// TIA Portal project "Water_Tank_For_Exam" (V12)

(* hardware
DEVICE "S7-1200 station_1"  SIMATIC 1200-Station
   slot 0: "S7-1200 rack"  Rack  V1.0
   slot 1: "Water_Tank_Logic"  CPU 1211C DC/DC/DC  6ES7 211-1AE31-0XB0  V3.0
DEVICE "S7-1500 station_1"  S7-1500 station
   slot 0: "Rail_0"  6ES7 590-1***0-0AA0
   slot 1: "PLC_1"  CPU 1513-1 PN  6ES7 513-1AL00-0AB0  V1.0
   slot 2: "DI 16x24VDC HF_1"  DI 16x24VDC HF  6ES7 521-1BH00-0AB0  V1.0
   slot 3: "DQ 8x24VDC/2A HF_1"  DQ 8x24VDC/2A HF  6ES7 522-1BF00-0AB0  V1.0
*)

// ===== PLC "Water_Tank_Logic"  CPU 1211C DC/DC/DC =====

VAR_GLOBAL   // PLC tag table "Default tag table"
   "GreenValveOpenLED" AT %Q0.0 : Bool;
   "redTankEmpty" AT %Q0.1 : Bool;
   "YellowTankFull" AT %Q0.2 : Bool;
   "LowSensor" AT %I0.0 : Bool;
   "HighLSensor" AT %I0.1 : Bool;
   "Manual" AT %I0.2 : Bool;
   "start" AT %I0.3 : Bool;
   "detectContainer" AT %I0.4 : Bool;
   "waterValve" AT %Q0.4 : Bool;
   "lacth" AT %M0.0 : Bool;
   "OpenValvePB" AT %I0.5 : Bool;
   "flashingEmptyLED" AT %Q0.3 : Bool;
   "autoMode" AT %I0.6 : Bool;
   "Counter5Mem" AT %M100.1 : Bool;
   "TimerFlash" AT %M100.0 : Bool;
   "Tag_1" AT %M100.2 : Bool;
END_VAR

// folder: System blocks/Program resources

DATA_BLOCK "IEC_Timer_0_DB"   // DB1
{ S7_Optimized_Access := 'FALSE' }
AUTHOR : Simatic
FAMILY : IEC
NAME : IEC_TMR
VERSION : 1.0
// stored: InstanceOfName ?
"?"
BEGIN
END_DATA_BLOCK

DATA_BLOCK "Counter_5"   // DB2
{ S7_Optimized_Access := 'FALSE' }
AUTHOR : Simatic
FAMILY : IEC
NAME : CNTR
VERSION : 1.0
// stored: InstanceOfName ?
"?"
BEGIN
END_DATA_BLOCK

DATA_BLOCK "Water_Running_timer"   // DB3
{ S7_Optimized_Access := 'FALSE' }
AUTHOR : Simatic
FAMILY : IEC
NAME : IEC_TMR
VERSION : 1.0
// stored: InstanceOfName ?
"?"
BEGIN
END_DATA_BLOCK

DATA_BLOCK "water_Still_in_Tank"   // DB4
{ S7_Optimized_Access := 'FALSE' }
AUTHOR : Simatic
FAMILY : IEC
NAME : IEC_TMR
VERSION : 1.0
// stored: InstanceOfName ?
"?"
BEGIN
END_DATA_BLOCK

DATA_BLOCK "Valve_counter"   // DB5
{ S7_Optimized_Access := 'FALSE' }
AUTHOR : Simatic
FAMILY : IEC
NAME : CNTR
VERSION : 1.0
// stored: InstanceOfName ?
"?"
BEGIN
END_DATA_BLOCK

DATA_BLOCK "Pulsating"   // DB7
{ S7_Optimized_Access := 'FALSE' }
AUTHOR : Simatic
FAMILY : IEC
NAME : IEC_TMR
VERSION : 1.0
// stored: InstanceOfName ?
"?"
BEGIN
END_DATA_BLOCK

DATA_BLOCK "Water_Valve_Timer"   // DB8
{ S7_Optimized_Access := 'FALSE' }
AUTHOR : Simatic
FAMILY : IEC
NAME : IEC_TMR
VERSION : 1.0
// stored: InstanceOfName ?
"?"
BEGIN
END_DATA_BLOCK

DATA_BLOCK "Water_remaining_timer"   // DB9
{ S7_Optimized_Access := 'FALSE' }
AUTHOR : Simatic
FAMILY : IEC
NAME : IEC_TMR
VERSION : 1.0
// stored: InstanceOfName ?
"?"
BEGIN
END_DATA_BLOCK

// folder: (top level)

FUNCTION "Water_Tank_Status_And_Control" : Void   // FC1, LAD
{ S7_Optimized_Access := 'FALSE' }
VERSION : 0.1
BEGIN

REGION Network 1: LED to indicate a low tank
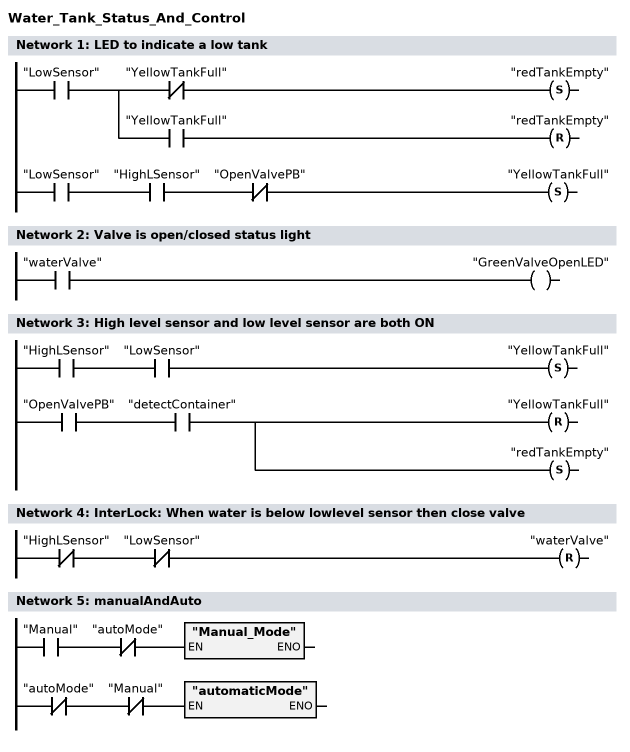
   RUNG wire#powerrail
      Contact( "LowSensor" )
      wire#w1
      I_Contact( "YellowTankFull" )
      S_Coil( "redTankEmpty" )
   END_RUNG
   RUNG wire#w1
      Contact( "YellowTankFull" )
      R_Coil( "redTankEmpty" )
   END_RUNG
   RUNG wire#powerrail
      Contact( "LowSensor" )
      Contact( "HighLSensor" )
      I_Contact( "OpenValvePB" )
      S_Coil( "YellowTankFull" )
   END_RUNG
   // the same network as SCL:
   IF "LowSensor" AND NOT "YellowTankFull" THEN "redTankEmpty" := TRUE; END_IF;
   IF "LowSensor" AND "YellowTankFull" THEN "redTankEmpty" := FALSE; END_IF;
   IF "LowSensor" AND "HighLSensor" AND NOT "OpenValvePB" THEN "YellowTankFull" := TRUE; END_IF;
END_REGION

REGION Network 2: Valve is open/closed status light
   RUNG wire#powerrail
      Contact( "waterValve" )
      Coil( "GreenValveOpenLED" )
   END_RUNG
   // the same network as SCL:
   "GreenValveOpenLED" := "waterValve";
END_REGION

REGION Network 3: High level sensor and low level sensor are both ON
   RUNG wire#powerrail
      Contact( "HighLSensor" )
      Contact( "LowSensor" )
      S_Coil( "YellowTankFull" )
   END_RUNG
   RUNG wire#powerrail
      Contact( "OpenValvePB" )
      Contact( "detectContainer" )
      wire#w1
      R_Coil( "YellowTankFull" )
   END_RUNG
   RUNG wire#w1
      S_Coil( "redTankEmpty" )
   END_RUNG
   // the same network as SCL:
   IF "HighLSensor" AND "LowSensor" THEN "YellowTankFull" := TRUE; END_IF;
   IF "OpenValvePB" AND "detectContainer" THEN
       "YellowTankFull" := FALSE;
       "redTankEmpty" := TRUE;
   END_IF;
END_REGION

REGION Network 4: InterLock: When water is below lowlevel sensor then close valve
   RUNG wire#powerrail
      I_Contact( "HighLSensor" )
      I_Contact( "LowSensor" )
      R_Coil( "waterValve" )
   END_RUNG
   // the same network as SCL:
   IF NOT "HighLSensor" AND NOT "LowSensor" THEN "waterValve" := FALSE; END_IF;
END_REGION

REGION Network 5: manualAndAuto
   RUNG wire#powerrail
      Contact( "Manual" )
      I_Contact( "autoMode" )
      "Manual_Mode"()
   END_RUNG
   RUNG wire#powerrail
      I_Contact( "autoMode" )
      I_Contact( "Manual" )
      "automaticMode"()
   END_RUNG
   // the same network as SCL:
   IF "Manual" AND NOT "autoMode" THEN "Manual_Mode"(); END_IF;
   IF NOT "autoMode" AND NOT "Manual" THEN "automaticMode"(); END_IF;
END_REGION
END_FUNCTION

FUNCTION "Manual_Mode" : Void   // FC2, LAD
{ S7_Optimized_Access := 'FALSE' }
VERSION : 0.1
   VAR_TEMP   // added for the SCL form of the ladder/FBD networks
      _w1 : Bool;
   END_VAR
BEGIN

REGION Network 1: manual mode
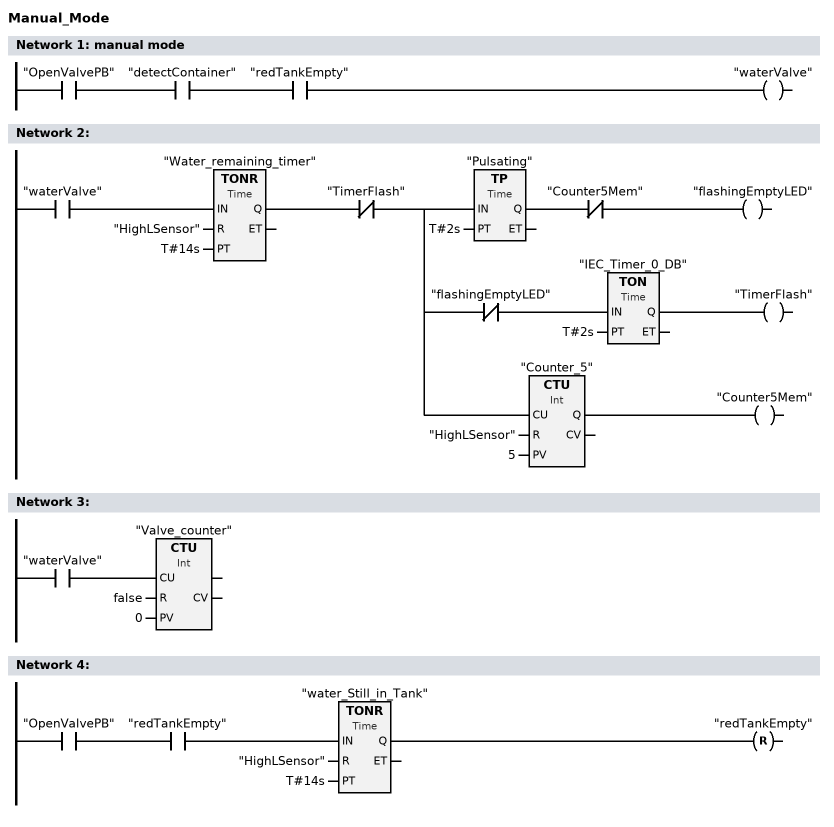
   RUNG wire#powerrail
      Contact( "OpenValvePB" )
      Contact( "detectContainer" )
      Contact( "redTankEmpty" )
      Coil( "waterValve" )
   END_RUNG
   // the same network as SCL:
   "waterValve" := "OpenValvePB" AND "detectContainer" AND "redTankEmpty";
END_REGION

REGION Network 2
   "Water_remaining_timer".TONR(IN := "waterValve", R := "HighLSensor", PT := T#14s);
   #_w1 := "Water_remaining_timer".Q AND NOT "TimerFlash";
   "Pulsating".TP(IN := #_w1, PT := T#2s);
   "flashingEmptyLED" := "Pulsating".Q AND NOT "Counter5Mem";
   "IEC_Timer_0_DB".TON(IN := #_w1 AND NOT "flashingEmptyLED", PT := T#2s);
   "TimerFlash" := "IEC_Timer_0_DB".Q;
   "Counter_5".CTU(CU := #_w1, R := "HighLSensor", PV := 5);
   "Counter5Mem" := "Counter_5".Q;
END_REGION

REGION Network 3
   "Valve_counter".CTU(CU := "waterValve", R := false, PV := 0);
END_REGION

REGION Network 4
   "water_Still_in_Tank".TONR(IN := "OpenValvePB" AND "redTankEmpty", R := "HighLSensor", PT := T#14s);
   IF "water_Still_in_Tank".Q THEN "redTankEmpty" := FALSE; END_IF;
END_REGION
END_FUNCTION

FUNCTION "automaticMode" : Void   // FC3, LAD
{ S7_Optimized_Access := 'FALSE' }
VERSION : 0.1
   VAR_TEMP   // added for the SCL form of the ladder/FBD networks
      _w1 : Bool;
   END_VAR
BEGIN

REGION Network 1: Automode Detects the container
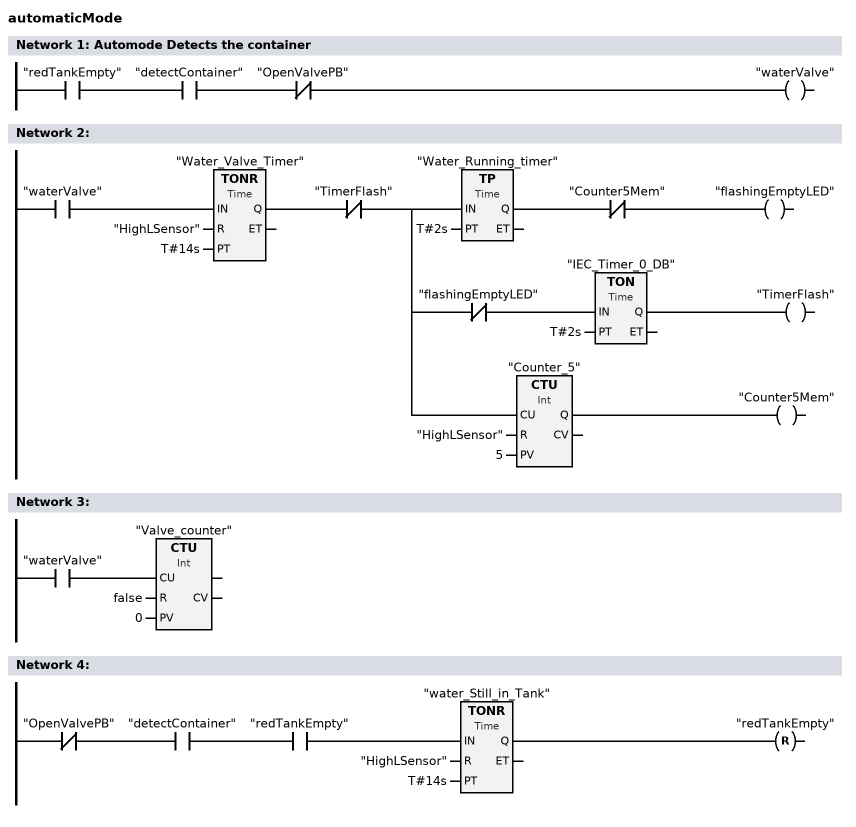
   RUNG wire#powerrail
      Contact( "redTankEmpty" )
      Contact( "detectContainer" )
      I_Contact( "OpenValvePB" )
      Coil( "waterValve" )
   END_RUNG
   // the same network as SCL:
   "waterValve" := "redTankEmpty" AND "detectContainer" AND NOT "OpenValvePB";
END_REGION

REGION Network 2
   "Water_Valve_Timer".TONR(IN := "waterValve", R := "HighLSensor", PT := T#14s);
   #_w1 := "Water_Valve_Timer".Q AND NOT "TimerFlash";
   "Water_Running_timer".TP(IN := #_w1, PT := T#2s);
   "flashingEmptyLED" := "Water_Running_timer".Q AND NOT "Counter5Mem";
   "IEC_Timer_0_DB".TON(IN := #_w1 AND NOT "flashingEmptyLED", PT := T#2s);
   "TimerFlash" := "IEC_Timer_0_DB".Q;
   "Counter_5".CTU(CU := #_w1, R := "HighLSensor", PV := 5);
   "Counter5Mem" := "Counter_5".Q;
END_REGION

REGION Network 3
   "Valve_counter".CTU(CU := "waterValve", R := false, PV := 0);
END_REGION

REGION Network 4
   "water_Still_in_Tank".TONR(IN := NOT "OpenValvePB" AND "detectContainer" AND "redTankEmpty",
                           R := "HighLSensor",
                           PT := T#14s);
   IF "water_Still_in_Tank".Q THEN "redTankEmpty" := FALSE; END_IF;
END_REGION
END_FUNCTION

ORGANIZATION_BLOCK "Main"   // OB1, LAD, ProgramCycle
TITLE = "Main Program Sweep (Cycle)"
{ S7_Optimized_Access := 'FALSE' }
VERSION : 0.1
   VAR_TEMP   // added for the SCL form of the ladder/FBD networks
      _w1 : Bool;
   END_VAR
BEGIN

REGION Network 1: Start and Stop the Whole plant
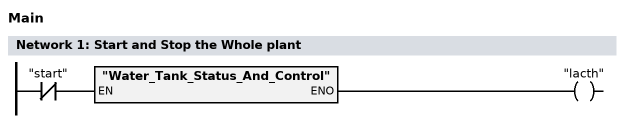
   RUNG wire#powerrail
      I_Contact( "start" )
      "Water_Tank_Status_And_Control"()
      Coil( "lacth" )
   END_RUNG
   // the same network as SCL:
   "Water_Tank_Status_And_Control"(EN := NOT "start", ENO => #_w1);
   "lacth" := #_w1;
END_REGION
END_ORGANIZATION_BLOCK

// ===== PLC "PLC_1"  CPU 1513-1 PN =====

VAR_GLOBAL   // PLC tag table "Default tag table"
   "delayR" AT %M100.0 : Bool;
   "Tag_1" AT %M100.1 : Bool;
END_VAR

VAR_GLOBAL   // PLC tag table "Default tag table_1"
   "GreenValveOpenLED" AT %Q0.0 : Bool;
   "redTankEmpty" AT %Q0.1 : Bool;
   "YellowTankFull" AT %Q0.2 : Bool;
   "LowSensor" AT %I0.0 : Bool;
   "HighLSensor" AT %I0.1 : Bool;
   "Manual" AT %I0.2 : Bool;
   "Stop" AT %I0.3 : Bool;
   "detectContainer" AT %I0.4 : Bool;
   "waterValve" AT %Q0.3 : Bool;
   "Start" AT %I0.5 : Bool;
   "lacth" AT %M0.0 : Bool;
   "OpenValvePB" AT %I0.6 : Bool;
   "flashingEmptyLED" AT %Q0.4 : Bool;
   "autoMode" AT %I0.7 : Bool;
END_VAR

VAR_GLOBAL CONSTANT   // PLC tag table "Default tag table_1"
   "OB_Main(1)" : OB_PCYCLE := 1;
END_VAR

// folder: System blocks/Program resources

DATA_BLOCK "IEC_Timer_0_DB_1"   // DB2
{ S7_Optimized_Access := 'FALSE' }
AUTHOR : Simatic
FAMILY : IEC
NAME : IEC_TMR
VERSION : 1.0
// stored: InstanceOfName ?
"?"
BEGIN
END_DATA_BLOCK

DATA_BLOCK "Water_Running_timer"   // DB3
{ S7_Optimized_Access := 'FALSE' }
AUTHOR : Simatic
FAMILY : IEC
NAME : IEC_TMR
VERSION : 1.0
// stored: InstanceOfName ?
"?"
BEGIN
END_DATA_BLOCK

DATA_BLOCK "Water_Draining_acc"   // DB4
{ S7_Optimized_Access := 'FALSE' }
AUTHOR : Simatic
FAMILY : IEC
NAME : IEC_TMR
VERSION : 1.0
// stored: InstanceOfName ?
"?"
BEGIN
END_DATA_BLOCK

DATA_BLOCK "Valve_counter"   // DB5
{ S7_Optimized_Access := 'FALSE' }
AUTHOR : Simatic
FAMILY : IEC
NAME : CNTR
VERSION : 1.0
// stored: InstanceOfName ?
"?"
BEGIN
END_DATA_BLOCK

DATA_BLOCK "IEC_Timer_0_DB_2"   // DB7
{ S7_Optimized_Access := 'FALSE' }
AUTHOR : Simatic
FAMILY : IEC
NAME : IEC_TMR
VERSION : 1.0
// stored: InstanceOfName ?
"?"
BEGIN
END_DATA_BLOCK

DATA_BLOCK "IEC_Counter_0_DB"   // DB8
{ S7_Optimized_Access := 'FALSE' }
AUTHOR : Simatic
FAMILY : IEC
NAME : CNTR
VERSION : 1.0
// stored: InstanceOfName ?
"?"
BEGIN
END_DATA_BLOCK

// folder: (top level)

FUNCTION "Water_Tank_Status_And_Control" : Void   // FC1, LAD
{ S7_Optimized_Access := 'FALSE' }
VERSION : 0.1
BEGIN

REGION Network 1: LED to indicate a low tank
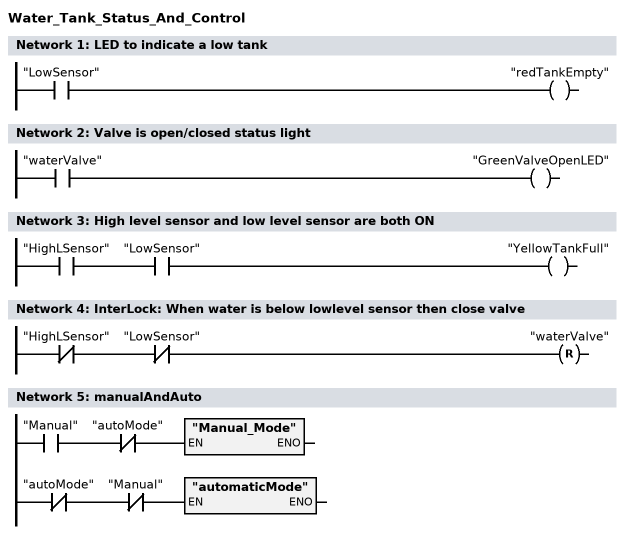
   RUNG wire#powerrail
      Contact( "LowSensor" )
      Coil( "redTankEmpty" )
   END_RUNG
   // the same network as SCL:
   "redTankEmpty" := "LowSensor";
END_REGION

REGION Network 2: Valve is open/closed status light
   RUNG wire#powerrail
      Contact( "waterValve" )
      Coil( "GreenValveOpenLED" )
   END_RUNG
   // the same network as SCL:
   "GreenValveOpenLED" := "waterValve";
END_REGION

REGION Network 3: High level sensor and low level sensor are both ON
   RUNG wire#powerrail
      Contact( "HighLSensor" )
      Contact( "LowSensor" )
      Coil( "YellowTankFull" )
   END_RUNG
   // the same network as SCL:
   "YellowTankFull" := "HighLSensor" AND "LowSensor";
END_REGION

REGION Network 4: InterLock: When water is below lowlevel sensor then close valve
   RUNG wire#powerrail
      I_Contact( "HighLSensor" )
      I_Contact( "LowSensor" )
      R_Coil( "waterValve" )
   END_RUNG
   // the same network as SCL:
   IF NOT "HighLSensor" AND NOT "LowSensor" THEN "waterValve" := FALSE; END_IF;
END_REGION

REGION Network 5: manualAndAuto
   RUNG wire#powerrail
      Contact( "Manual" )
      I_Contact( "autoMode" )
      "Manual_Mode"()
   END_RUNG
   RUNG wire#powerrail
      I_Contact( "autoMode" )
      I_Contact( "Manual" )
      "automaticMode"()
   END_RUNG
   // the same network as SCL:
   IF "Manual" AND NOT "autoMode" THEN "Manual_Mode"(); END_IF;
   IF NOT "autoMode" AND NOT "Manual" THEN "automaticMode"(); END_IF;
END_REGION
END_FUNCTION

FUNCTION "Manual_Mode" : Void   // FC2, LAD
{ S7_Optimized_Access := 'FALSE' }
VERSION : 0.1
   VAR_TEMP   // added for the SCL form of the ladder/FBD networks
      _w1 : Bool;
   END_VAR
BEGIN

REGION Network 1: manual mode
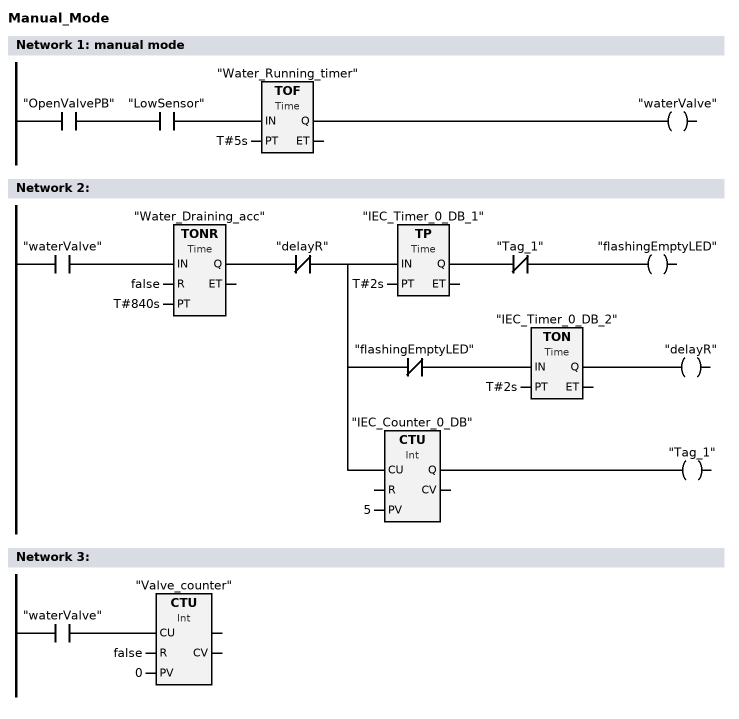
   "Water_Running_timer".TOF(IN := "OpenValvePB" AND "LowSensor", PT := T#5s);
   "waterValve" := "Water_Running_timer".Q;
END_REGION

REGION Network 2
   "Water_Draining_acc".TONR(IN := "waterValve", R := false, PT := T#840s);
   #_w1 := "Water_Draining_acc".Q AND NOT "delayR";
   "IEC_Timer_0_DB_1".TP(IN := #_w1, PT := T#2s);
   "flashingEmptyLED" := "IEC_Timer_0_DB_1".Q AND NOT "Tag_1";
   "IEC_Timer_0_DB_2".TON(IN := #_w1 AND NOT "flashingEmptyLED", PT := T#2s);
   "delayR" := "IEC_Timer_0_DB_2".Q;
   "IEC_Counter_0_DB".CTU(CU := #_w1, PV := 5);
   "Tag_1" := "IEC_Counter_0_DB".Q;
END_REGION

REGION Network 3
   "Valve_counter".CTU(CU := "waterValve", R := false, PV := 0);
END_REGION
END_FUNCTION

FUNCTION "automaticMode" : Void   // FC3, LAD
{ S7_Optimized_Access := 'FALSE' }
VERSION : 0.1
   VAR_TEMP   // added for the SCL form of the ladder/FBD networks
      _w1 : Bool;
   END_VAR
BEGIN

REGION Network 1: Automode Detects the container
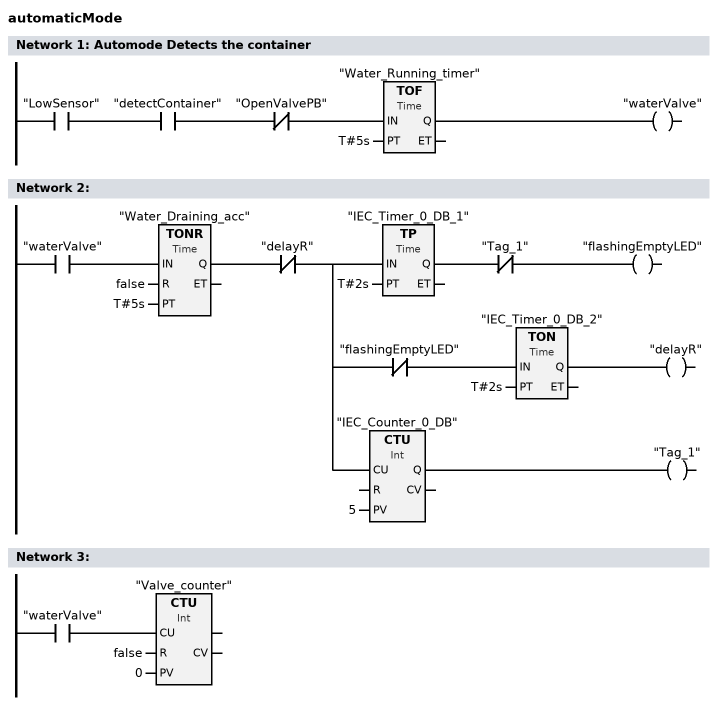
   "Water_Running_timer".TOF(IN := "LowSensor" AND "detectContainer" AND NOT "OpenValvePB", PT := T#5s);
   "waterValve" := "Water_Running_timer".Q;
END_REGION

REGION Network 2
   "Water_Draining_acc".TONR(IN := "waterValve", R := false, PT := T#5s);
   #_w1 := "Water_Draining_acc".Q AND NOT "delayR";
   "IEC_Timer_0_DB_1".TP(IN := #_w1, PT := T#2s);
   "flashingEmptyLED" := "IEC_Timer_0_DB_1".Q AND NOT "Tag_1";
   "IEC_Timer_0_DB_2".TON(IN := #_w1 AND NOT "flashingEmptyLED", PT := T#2s);
   "delayR" := "IEC_Timer_0_DB_2".Q;
   "IEC_Counter_0_DB".CTU(CU := #_w1, PV := 5);
   "Tag_1" := "IEC_Counter_0_DB".Q;
END_REGION

REGION Network 3
   "Valve_counter".CTU(CU := "waterValve", R := false, PV := 0);
END_REGION
END_FUNCTION

ORGANIZATION_BLOCK "Main"   // OB1, LAD, ProgramCycle
TITLE = "Main Program Sweep (Cycle)"
{ S7_Optimized_Access := 'FALSE' }
VERSION : 0.1
   VAR_INPUT
      Initial_Call : Bool;   // Initial call of this OB
      Remanence : Bool;   // =True, if remanent data are available
   END_VAR
   VAR_TEMP   // added for the SCL form of the ladder/FBD networks
      _w1 : Bool;
   END_VAR
BEGIN

REGION Network 1: Start and Stop the Whole plant
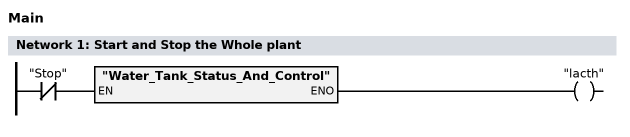
   RUNG wire#powerrail
      I_Contact( "Stop" )
      "Water_Tank_Status_And_Control"()
      Coil( "lacth" )
   END_RUNG
   // the same network as SCL:
   "Water_Tank_Status_And_Control"(EN := NOT "Stop", ENO => #_w1);
   "lacth" := #_w1;
END_REGION
END_ORGANIZATION_BLOCK